
FUNCTION CB_sel_dint : DINT


TITLE = ' Binary selection on 2 variables '
VERSION : '1.0'
AUTHOR  : CB
NAME    : sel_dint
FAMILY  : TNI

VAR_INPUT
    G : BOOL;
    IN0 : DINT ;
    IN1 : DINT ;

END_VAR

BEGIN

CB_sel_dint := SEL(G:= G, IN0 := IN0, IN1 := IN1);

END_FUNCTION
